% RSLogix 500 project training_two_setpoints_running_0.965.RSS, saved by version 8.30.00.16 %
PROJECT "UNTITLED"    % processor: Bul.1763 MicroLogix 1100 Series B %

PROGRAM FILES
  LAD 2 "MAIN"  3 rungs
  LAD 3 "FILTERDATA"  2 rungs
  LAD 4 "LOADCELLIN"  5 rungs
  LAD 5 "TRAINING"  8 rungs

DATA FILES
  O0 OUTPUT  4 elements
  I1 INPUT  6 elements
  S2 STATUS  66 elements
  B3 BINARY  3 elements
  T4 TIMER  2 elements
  C5 COUNTER  2 elements
  R6 CONTROL  1 elements
  N7 INTEGER  10 elements
  F8 FLOAT  10 elements

LADDER 2 "MAIN"
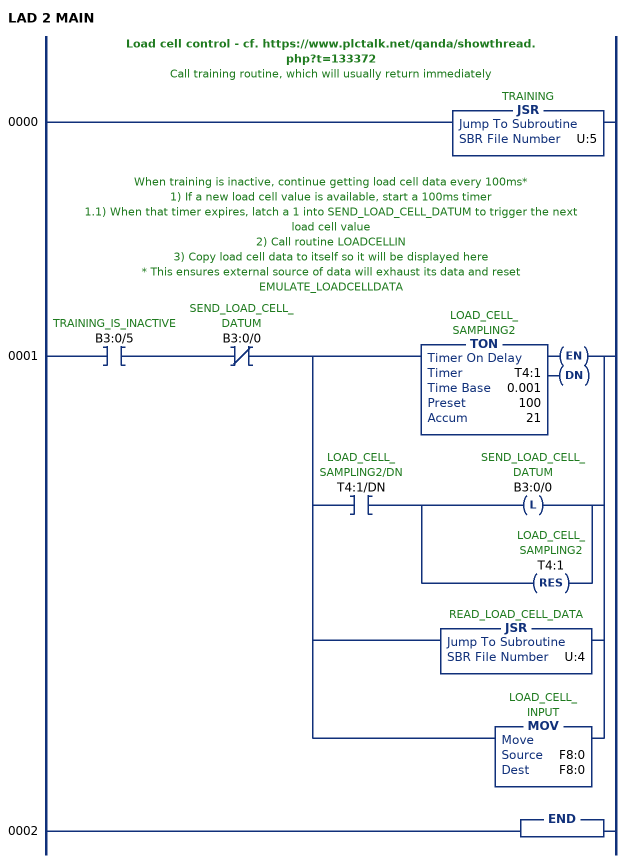
% Rung: 0 %
% TITLE: Load cell control - cf. https://www.plctalk.net/qanda/showthread.php?t=133372 %
% Call training routine, which will usually return immediately %
SOR JSR U:5 EOR
%   U:5  TRAINING %
% Rung: 1 %
% When training is inactive, continue getting load cell data every 100ms*
% 1) If a new load cell value is available, start a 100ms timer
% 1.1) When that timer expires, latch a 1 into SEND_LOAD_CELL_DATUM to trigger the next load cell value
% 2) Call routine LOADCELLIN
% 3) Copy load cell data to itself so it will be displayed here
% * This ensures external source of data will exhaust its data and reset EMULATE_LOADCELLDATA %
SOR XIC B3:0/5 XIO B3:0/0 BST BST TON T4:1 0.001 100 21 NXB XIC T4:1/DN BST OTL B3:0/0 NXB RES T4:1 BND BND NXB JSR U:4 NXB MOV F8:0 F8:0 BND EOR
%   B3:0/5  TRAINING_IS_INACTIVE %
%   B3:0/0  SEND_LOAD_CELL_DATUM %
%   T4:1  LOAD_CELL_SAMPLING2 %
%   U:4  READ_LOAD_CELL_DATA %
%   F8:0  LOAD_CELL_INPUT %
% Rung: 2 %
SOR END EOR

LADDER 3 "FILTERDATA"
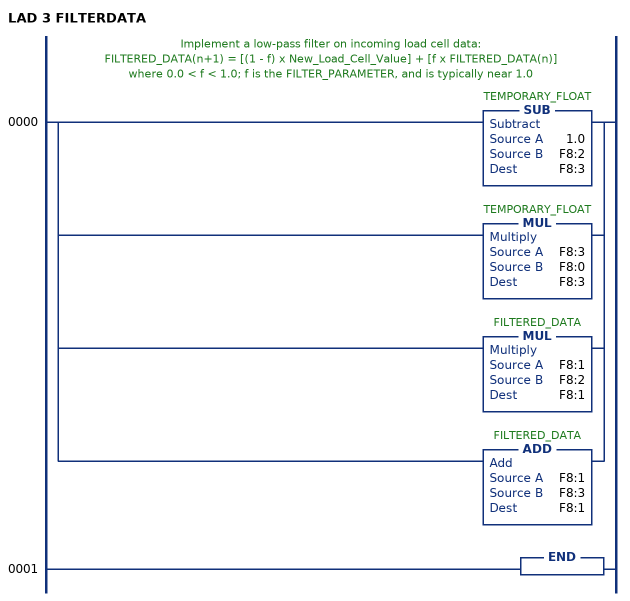
% Rung: 0 %
% Implement a low-pass filter on incoming load cell data:
% 
%   FILTERED_DATA(n+1) = [(1 - f) x New_Load_Cell_Value] + [f x FILTERED_DATA(n)]
% 
% where 0.0 < f < 1.0; f is the FILTER_PARAMETER, and is typically near 1.0 %
SOR BST SUB 1.0 F8:2 F8:3 NXB MUL F8:3 F8:0 F8:3 NXB MUL F8:1 F8:2 F8:1 NXB ADD F8:1 F8:3 F8:1 BND EOR
%   F8:2  FILTER_PARAMETER %
%   F8:3  TEMPORARY_FLOAT %
%   F8:0  LOAD_CELL_INPUT %
%   F8:1  FILTERED_DATA %
% Rung: 1 %
SOR END EOR

LADDER 4 "LOADCELLIN"
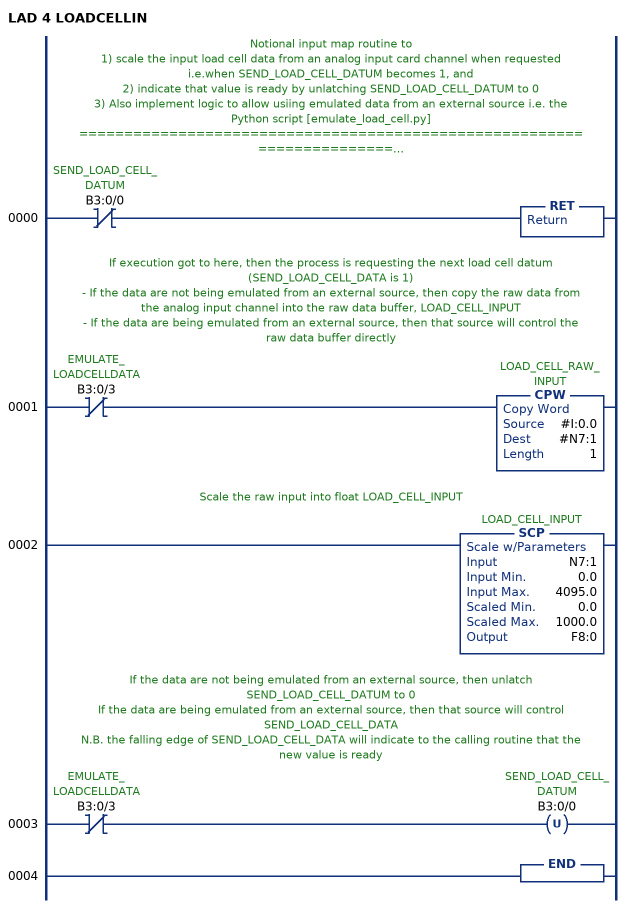
% Rung: 0 %
% Notional input map routine to
% 1) scale the input load cell data from an analog input card channel when requested i.e.when SEND_LOAD_CELL_DATUM becomes 1, and
% 2) indicate that value is ready by unlatching SEND_LOAD_CELL_DATUM to 0
% 3) Also implement logic to allow usiing emulated data from an external source i.e. the Python script [emulate_load_cell.py]
% 
% ========================================================================
% If SEND_LOAD_CELL_DATA is 0 i.e. not 1, then return and do nothing %
SOR XIO B3:0/0 RET EOR
%   B3:0/0  SEND_LOAD_CELL_DATUM %
% Rung: 1 %
% If execution got to here, then the process is requesting the next load cell datum (SEND_LOAD_CELL_DATA is 1)
% - If the data are not being emulated from an external source, then copy the raw data from the analog input channel into the raw data buffer, LOAD_CELL_INPUT
% - If the data are being emulated from an external source, then that source will control the raw data buffer directly %
SOR XIO B3:0/3 CPW #I:0.0 #N7:1 1 EOR
%   B3:0/3  EMULATE_LOADCELLDATA %
%   N7:1  LOAD_CELL_RAW_INPUT %
% Rung: 2 %
% Scale the raw input into float LOAD_CELL_INPUT %
SOR SCP N7:1 0.0 4095.0 0.0 1000.0 F8:0 EOR
%   N7:1  LOAD_CELL_RAW_INPUT %
%   F8:0  LOAD_CELL_INPUT %
% Rung: 3 %
% If the data are not being emulated from an external source, then unlatch SEND_LOAD_CELL_DATUM to 0
% If the data are being emulated from an external source, then that source will control SEND_LOAD_CELL_DATA
% N.B. the falling edge of SEND_LOAD_CELL_DATA will indicate to the calling routine that the new value is ready %
SOR XIO B3:0/3 OTU B3:0/0 EOR
%   B3:0/3  EMULATE_LOADCELLDATA %
%   B3:0/0  SEND_LOAD_CELL_DATUM %
% Rung: 4 %
SOR END EOR

LADDER 5 "TRAINING"
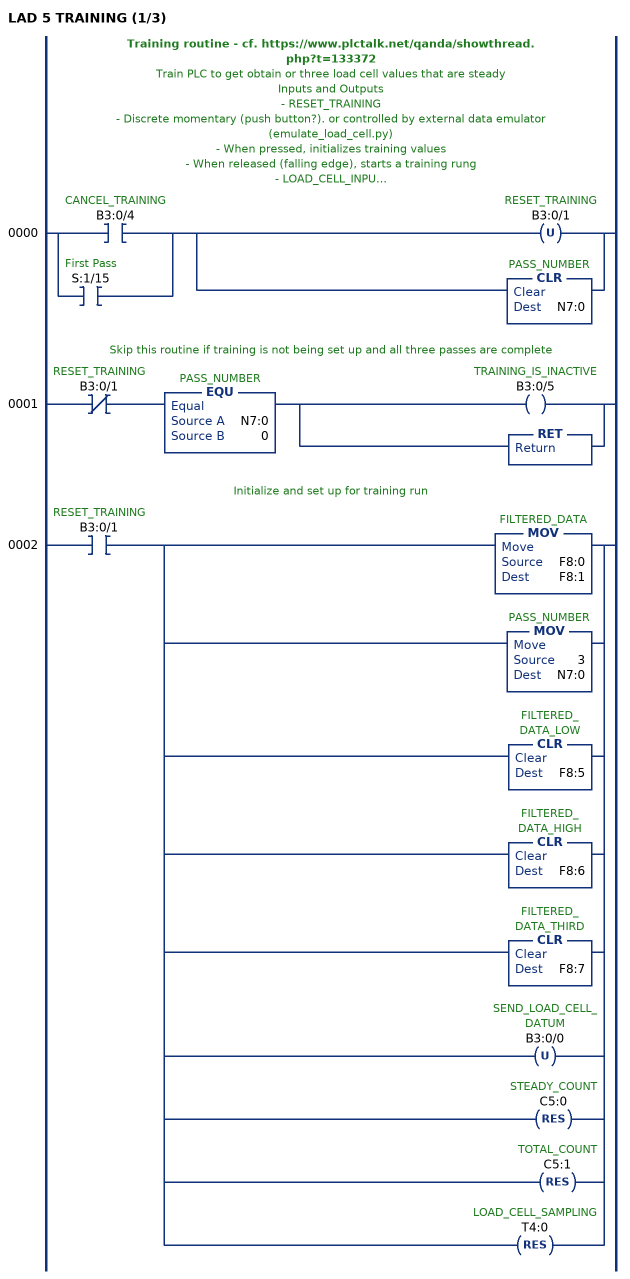
% Rung: 0 %
% TITLE: Training routine - cf. https://www.plctalk.net/qanda/showthread.php?t=133372 %
% Train PLC to get obtain or three load cell values that are steady
% 
% Inputs and Outputs
% - RESET_TRAINING
%   - Discrete momentary (push button?). or controlled by external data emulator (emulate_load_cell.py)
%   - When pressed, initializes training values
%   - When released (falling edge), starts a training rung
% - LOAD_CELL_INPUT
%   - Analog float value that is loaded from load cell in response to a rising edge of Boolean SEND_LOAD_CELL_DATUM
% - SEND_LOAD_CELL_DATUM (both output-ish and input-ish)
%   - Output:  written to as a 1 by this routine to indicate 100ms have expired and it is time for the next load cell value
%   - Input:  written to as a 0 by another entity to after putting a new value into LOAD_CELL_INPUT
%     - This falling edge indicates a new LOAD_CELL_INPUT is ready
%     - The other entity could be an I/O mapping routine, or the Python script [emulate_load_cell.py]
% 
% ========================================================================
% First rung:  respond to request to cancel training %
SOR BST XIC B3:0/4 NXB XIC S:1/15 BND BST OTU B3:0/1 NXB CLR N7:0 BND EOR
%   B3:0/4  CANCEL_TRAINING %
%   S:1/15  "First Pass" %
%   B3:0/1  RESET_TRAINING %
%   N7:0  PASS_NUMBER %
% Rung: 1 %
% Skip this routine if training is not being set up and all three passes are complete %
SOR XIO B3:0/1 EQU N7:0 0 BST OTE B3:0/5 NXB RET BND EOR
%   B3:0/1  RESET_TRAINING %
%   N7:0  PASS_NUMBER %
%   B3:0/5  TRAINING_IS_INACTIVE %
% Rung: 2 %
% Initialize and set up for training run %
SOR XIC B3:0/1 BST MOV F8:0 F8:1 NXB MOV 3 N7:0 NXB CLR F8:5 NXB CLR F8:6 NXB CLR F8:7 NXB OTU B3:0/0 NXB RES C5:0 NXB RES C5:1 NXB RES T4:0 BND EOR
%   B3:0/1  RESET_TRAINING %
%   F8:0  LOAD_CELL_INPUT %
%   F8:1  FILTERED_DATA %
%   N7:0  PASS_NUMBER %
%   F8:5  FILTERED_DATA_LOW %
%   F8:6  FILTERED_DATA_HIGH %
%   F8:7  FILTERED_DATA_THIRD %
%   B3:0/0  SEND_LOAD_CELL_DATUM %
%   C5:0  STEADY_COUNT %
%   C5:1  TOTAL_COUNT %
%   T4:0  LOAD_CELL_SAMPLING %

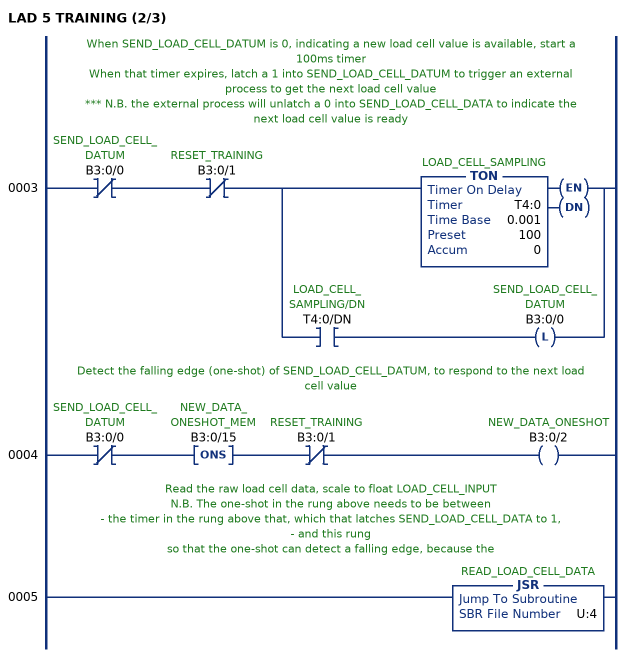
% Rung: 3 %
% When SEND_LOAD_CELL_DATUM is 0, indicating a new load cell value is available, start a 100ms timer
% When that timer expires, latch a 1 into SEND_LOAD_CELL_DATUM to trigger an external process to get the next load cell value
% *** N.B. the external process will unlatch a 0 into SEND_LOAD_CELL_DATA to indicate the next load cell value is ready %
SOR XIO B3:0/0 XIO B3:0/1 BST TON T4:0 0.001 100 0 NXB XIC T4:0/DN OTL B3:0/0 BND EOR
%   B3:0/0  SEND_LOAD_CELL_DATUM %
%   B3:0/1  RESET_TRAINING %
%   T4:0  LOAD_CELL_SAMPLING %
% Rung: 4 %
% Detect the falling edge (one-shot) of SEND_LOAD_CELL_DATUM, to respond to the next load cell value %
SOR XIO B3:0/0 ONS B3:0/15 XIO B3:0/1 OTE B3:0/2 EOR
%   B3:0/0  SEND_LOAD_CELL_DATUM %
%   B3:0/15  NEW_DATA_ONESHOT_MEM %
%   B3:0/1  RESET_TRAINING %
%   B3:0/2  NEW_DATA_ONESHOT %
% Rung: 5 %
% Read the raw load cell data, scale to float LOAD_CELL_INPUT
% 
% N.B. The one-shot in the rung above needs to be between
%         - the timer in the rung above that, which that latches SEND_LOAD_CELL_DATA to 1,
%         - and this rung
%         so that the one-shot can detect a falling edge, because the %
SOR JSR U:4 EOR
%   U:4  READ_LOAD_CELL_DATA %

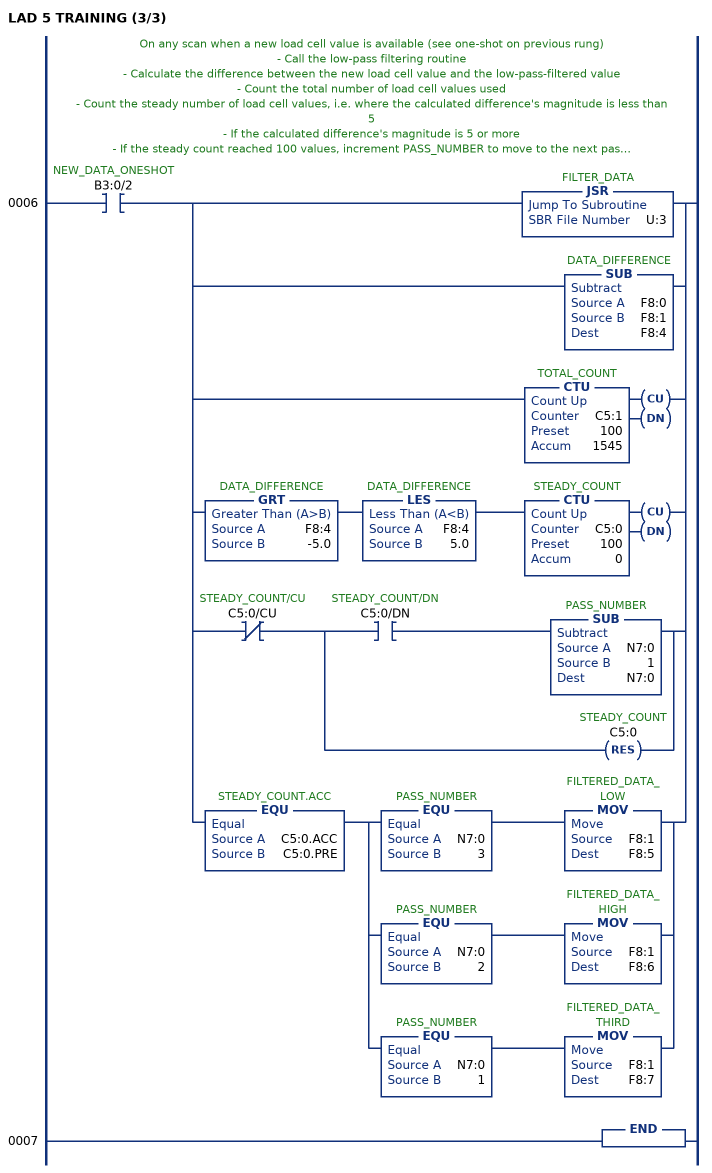
% Rung: 6 %
% On any scan when a new load cell value is available (see one-shot on previous rung)
% - Call the low-pass filtering routine
% - Calculate the difference between the new load cell value and the low-pass-filtered value
% - Count the total number of load cell values used
% - Count the steady number of load cell values, i.e. where the calculated difference's magnitude is less than 5
% - If the calculated difference's magnitude is 5 or more
%   - If the steady count reached 100 values, increment PASS_NUMBER to move to the next pass
%   - Clear the steady count
% - On the scan when the steady count reaches 100, save the current filtered value to the float of the current pass %
SOR XIC B3:0/2 BST JSR U:3 NXB SUB F8:0 F8:1 F8:4 NXB CTU C5:1 100 1545 NXB GRT F8:4 -5.0 LES F8:4 5.0 CTU C5:0 100 0 NXB XIO C5:0/CU BST XIC C5:0/DN SUB N7:0 1 N7:0 NXB RES C5:0 BND NXB EQU C5:0.ACC C5:0.PRE BST EQU N7:0 3 MOV F8:1 F8:5 NXB EQU N7:0 2 MOV F8:1 F8:6 NXB EQU N7:0 1 MOV F8:1 F8:7 BND BND EOR
%   B3:0/2  NEW_DATA_ONESHOT %
%   U:3  FILTER_DATA %
%   F8:0  LOAD_CELL_INPUT %
%   F8:1  FILTERED_DATA %
%   F8:4  DATA_DIFFERENCE %
%   C5:1  TOTAL_COUNT %
%   C5:0  STEADY_COUNT %
%   N7:0  PASS_NUMBER %
%   F8:5  FILTERED_DATA_LOW %
%   F8:6  FILTERED_DATA_HIGH %
%   F8:7  FILTERED_DATA_THIRD %
% Rung: 7 %
SOR END EOR

DATA TABLE (non-zero values as saved)
DATA B3
% B3:0 % 0X8024 0X0000 0X0000
DATA T4
% .PRE .ACC %
% T4:0 % 100 0
% T4:1 % 100 21
DATA C5
% .PRE .ACC %
% C5:0 % 100 0
% C5:1 % 100 1545
DATA R6
% .LEN .POS %
% R6:0 % 16 0
DATA F8
% F8:0 % 0 182.7578 0.965 6.196586 -5.712646
% F8:5 % 184.5199 273.3434 183.8225 0 0
